INTERFACE ITF_SPM_HMI_Lacznik EXTENDS B_Baza.ITF_PodzespolBazowy_HMI_Lacznik

END_INTERFACE

(* stored: Version 1.1.0.1
   Itf ITF_SPM_HMI_Lacznik: Id {8a699414-7eaf-4b79-8e49-986bb1b2576e} *)
